{attribute 'linkalways'} 
{attribute 'no_explicit_call' := 'This FB is a CLASS and must be accessed using methods or properties'}
{attribute 'enable_dynamic_creation'}
FUNCTION_BLOCK Node_F_VN_FillContainerExp_TcVnVector4_LREAL EXTENDS VisionNode
VAR
    ipContainer : _ITcVnContainer;
    aValue : _TcVnVector4_LREAL;
    nStartIdx : _ULINT(0);
    nCount : _ULINT(0);
    hrPrev : _HRESULT(S_OK);
    hresult : _HRESULT(S_OK);
END_VAR

METHOD PUBLIC  Clone : I_Node
VAR
    pNode : POINTER TO Node_F_VN_FillContainerExp_TcVnVector4_LREAL;
END_VAR
pNode := __NEW(Node_F_VN_FillContainerExp_TcVnVector4_LREAL);
Clone := pNode^;
END_METHOD

METHOD FB_init : BOOL
VAR_INPUT
    bInitRetains : BOOL; // if TRUE, the retain variables are initialized (warm start / cold start)
    bInCopyCode : BOOL;  // if TRUE, the instance afterwards gets moved into the copy code (online change)
END_VAR
AddInput('ipContainer', ipContainer);
AddInput('aValue', aValue);
AddInput('nStartIdx', nStartIdx);
AddInput('nCount', nCount);
AddInput('hrPrev', hrPrev);
AddOutput('ipContainer', ipContainer);
AddOutput('hresult',hresult);
END_METHOD

METHOD PROTECTED OnExecute : HRESULT
hresult.Value := F_VN_FillContainerExp_TcVnVector4_LREAL(
    ipContainer := ipContainer.Value,
    aValue := aValue.Value,
    nStartIdx := nStartIdx.Value,
    nCount := nCount.Value,
    hrPrev:= hrPrev.Value);
END_METHOD

METHOD PUBLIC PreExecutionCheck
VAR_INPUT
    Check : I_PreExecutionChecks;
END_VAR
Check.IsTrue(ipContainer.IsValid, 'ipContainer must be a valid container');
Check.IsTrue(ipContainer.HasType(TC_GLOBAL_CONST_LIST.ContainerType_Vector_TcVnVector4_LREAL), 'ipContainer contains incorrect type');
END_METHOD

END_FUNCTION_BLOCK

(* stored: Version 1.1.0.1, ProductVersion 3.1.4024.13
   POU Node_F_VN_FillContainerExp_TcVnVector4_LREAL: Id {e454a02a-3f97-4c26-bcbf-9b1a4659149d}, SpecialFunc None
   Folder Constructor: Id {309b0875-b53c-4efb-a9e9-c4f1eec6c378}
   Method Clone: Id {80cedff3-d4f5-4d79-b9f3-ba737d6f7c42}
   Method FB_init: Id {a9dd6128-e2a8-4574-98eb-91ad6c9d59c8}
   Method OnExecute: Id {abbee4f8-013d-4834-a6ea-cd959a8f6b77}
   Method PreExecutionCheck: Id {f05431db-3e94-4069-b3ac-ab1e319e3267} *)
